FUNCTION_BLOCK FB_SimBarcodeScanner EXTENDS FB_SimStation
VAR_INPUT
END_VAR
VAR_OUTPUT
END_VAR
VAR
	rand						: DRAND;
	tmrWork						: TON;
	sBarcode					: STRING(255);
END_VAR

METHOD PROTECTED  DoWork : BOOL
VAR_INPUT
END_VAR
rand(Seed:=777);
tmrWork(IN:=TRUE, PT:=T#3S);
IF tmrWork.Q THEN
	sBarcode := CONCAT('BRCD', TO_STRING(TO_DINT(rand.Num * 10000)));
	tmrWork(IN:=FALSE);
	DoWork := TRUE;
END_IF
END_METHOD

METHOD PROTECTED  UpdatePartStatus : PVOID
VAR_INPUT
END_VAR
IF pPartStatus <> 0 THEN
	pPartStatus^.bBarcodeStatus := TRUE;
	pPartStatus^.sBarcode := sBarcode;
END_IF
END_METHOD

END_FUNCTION_BLOCK

(* stored: Version 1.1.0.1, ProductVersion 3.1.4024.12
   POU FB_SimBarcodeScanner: Id {aaabbb18-d528-4ab4-a05e-daf444c77711}, SpecialFunc None
   Method DoWork: Id {590a7327-f3eb-4471-a88f-0b554007160f}
   Method UpdatePartStatus: Id {6bb335b6-c98f-49c7-a83c-0c6714d37d29} *)
